{attribute 'linkalways'} 
{attribute 'no_explicit_call' := 'This FB is a CLASS and must be accessed using methods or properties'}
{attribute 'enable_dynamic_creation'}
FUNCTION_BLOCK Node_ContainerType_Vector_Vector_TcVnDMatch EXTENDS Node
VAR
    out : _GUID;
END_VAR

METHOD PUBLIC  Clone : I_Node
VAR
	pNode : POINTER TO Node_ContainerType_Vector_Vector_TcVnDMatch;
END_VAR
pNode := __NEW(Node_ContainerType_Vector_Vector_TcVnDMatch);
Clone := pNode^;
END_METHOD

METHOD FB_init : BOOL
VAR_INPUT
	bInitRetains : BOOL; // if TRUE, the retain variables are initialized (warm start / cold start)
	bInCopyCode : BOOL;  // if TRUE, the instance afterwards gets moved into the copy code (online change)
END_VAR
AddOutput('out', out);
END_METHOD

METHOD PROTECTED OnExecute
out.Value := ContainerType_Vector_Vector_TcVnDMatch;
END_METHOD

END_FUNCTION_BLOCK

(* stored: Version 1.1.0.1, ProductVersion 3.1.4026.17
   POU Node_ContainerType_Vector_Vector_TcVnDMatch: Id {85e01546-fac2-0cbe-0330-590afd4818e5}, SpecialFunc None
   Folder Constructor: Id {47e94eb9-1bf1-09a3-0e1e-5ba6a1abd06e}
   Method Clone: Id {5b066aee-cce4-0976-0a3d-c3f93ce812f3}
   Method FB_init: Id {15727831-71a2-0c71-03cf-a2ed83c59ea4}
   Method OnExecute: Id {064fd5ab-e5ae-0bdd-25f7-68722381ad3e} *)
